FUNCTION_BLOCK CU020AutomatParalell_1_Task EXTENDS TcoTaskedSequencer 

VAR
	_customTimer: TON;
END_VAR

Run();

(*~
	<docu>
		<summary>
			Main method of the sequener. Custom code needs to be placed here. The sequencer is executed by call of **Instance.Run()** method.
			This method is abstract, and it must be overridden in derived block.
		</summary>
	</docu>
~*)
METHOD PROTECTED Main : BOOL
// Takes mode (step/continous) from the parent controller
THIS^.ModeController.Mode := ParentSequence.ModeController.Mode;

IF (Step(1000, TRUE, 'PARALELL STEP - EXAMPLE OF TIMERS')) THEN
    //-------------------------------------    
		StepCompleteWhen(CurrentStep.Duration >= T#300mS);	
    //-------------------------------------
END_IF
IF (Step(1100, TRUE, 'PARALELL STEP - EXAMPLE OF TIMERS')) THEN
    //-------------------------------------    
		StepCompleteWhen(inCondition:=Timer_1(TRUE,T#100MS));	
    //-------------------------------------
END_IF
IF (Step(1200, TRUE, 'PARALELL STEP - EXAMPLE OF TIMERS')) THEN
    //-------------------------------------    
		StepCompleteWhen(inCondition:=Timer_1(TRUE,T#200MS));	
    //-------------------------------------
END_IF


IF THIS^.IsFreshState THEN
	_customTimer(IN:=FALSE);
END_IF
IF (Step(1300, TRUE, 'PARALELL STEP - EXAMPLE OF TIMERS')) THEN
    //-------------------------------------    

		_customTimer(IN:=TRUE,PT:=T#200MS);
		StepCompleteWhen(inCondition:=_customTimer.Q);	
    //-------------------------------------
END_IF


IF (Step(10000, TRUE, 'PARALELL TASK DONE')) THEN
    //-------------------------------------
    _task.DoneWhen(TRUE );
    //-------------------------------------	
END_IF
END_METHOD

PROPERTY ParentSequence : REFERENCE TO CU020AutomatTask
GET
VAR
    _parentSequence : POINTER TO CU020AutomatTask;
END_VAR
IF __QUERYPOINTER(Parent, _parentSequence) THEN 
    ParentSequence REF= _parentSequence^;              
END_IF
END_GET
END_PROPERTY

END_FUNCTION_BLOCK

(* stored: Version 1.1.0.1
   POU CU020AutomatParalell_1_Task: Id {7dce8988-4b2b-4216-8f19-55921a520122}, SpecialFunc None
   Method Main: Id {483b5000-d54a-4421-a56c-2043f42afb90}
   Property ParentSequence: Id {1d0d157e-843a-44ea-9393-c780dd43c67c}
   Get Get: Id {e34b7924-2f1c-4f2b-8b01-7a6802702a95} *)
